// TIA Portal project "pick and place 3 things" (V16)
// Vorlageprojekt für das Buch mit Zielsystem S7-1200

(* hardware
DEVICE "S7-1200-Station_1"  S7-1200 Station
   slot 0: "Baugruppenträger_0"  Rack  V1.0
   slot 1: "PLC_1"  CPU 1211C DC/DC/DC  6ES7 211-1AE40-0XB0  V4.1
*)

// ===== PLC "PLC_1"  CPU 1211C DC/DC/DC =====

VAR_GLOBAL   // PLC tag table "Standard-Variablentabelle"
   "start" AT %I0.0 : Bool;
   "conv" AT %Q0.0 : Bool;
   "emitter" AT %Q0.1 : Bool;
   "z down" AT %Q0.2 : Bool;
   "grab" AT %Q0.3 : Bool;
   "z sensor" AT %I0.1 : Bool;
   "diffuse sens" AT %I0.2 : Bool;
   "diffuse sens memory" AT %M0.0 : Bool;
   "box detecd" AT %I0.3 : Bool;
   "box detecd memory" AT %M0.1 : Bool;
   "grab memory" AT %M0.2 : Bool;
   "z sens memory" AT %M0.3 : Bool;
   "x move" AT %Q0.4 : Bool;
   "x sensor" AT %I0.4 : Bool;
   "x sens memory\" AT %M0.4 : Bool;
   "Tag_1" AT %M0.5 : Bool;
   "Tag_2" AT %M0.7 : Bool;
   "set for timer1" AT %M1.0 : Bool;
   "Tag_4" AT %M1.1 : Bool;
   "Tag_5" AT %M1.2 : Bool;
   "set for timer 2" AT %M1.3 : Bool;
   "conv2" AT %Q0.5 : Bool;
   "diffues2" AT %I0.5 : Bool;
   "Tag_7" AT %M0.6 : Bool;
   "emitter2" AT %Q0.6 : Bool;
   "counter" AT %M1.4 : Bool;
   "Tag_9" AT %M1.5 : Bool;
   "Tag_10" AT %M1.6 : Bool;
   "Tag_8" AT %M2.0 : Bool;
   "sr for counter" AT %M2.1 : Bool;
   "reset for counter sr" AT %M2.2 : Bool;
   "stop" AT %I0.6 : Bool;
   "Tag_13" AT %M2.5 : Bool;
   "Tag_14" AT %M3.1 : Bool;
END_VAR

// folder: System blocks/Program resources

DATA_BLOCK "IEC_Timer_0_DB"   // DB1
{ S7_Optimized_Access := 'TRUE' }
AUTHOR : Simatic
FAMILY : IEC
NAME : IEC_TMR
VERSION : 1.0
// stored: InstanceOfName IEC_TIMER
"IEC_TIMER"
BEGIN
END_DATA_BLOCK

DATA_BLOCK "IEC_Timer_0_DB_1"   // DB2
{ S7_Optimized_Access := 'TRUE' }
AUTHOR : Simatic
FAMILY : IEC
NAME : IEC_TMR
VERSION : 1.0
// stored: InstanceOfName IEC_TIMER
"IEC_TIMER"
BEGIN
END_DATA_BLOCK

DATA_BLOCK "IEC_Counter_0_DB"   // DB3
{ S7_Optimized_Access := 'TRUE' }
AUTHOR : Simatic
FAMILY : IEC
NAME : CNTR
VERSION : 1.0
// stored: InstanceOfName IEC_COUNTER
"IEC_COUNTER"
BEGIN
END_DATA_BLOCK

// folder: (top level)

FUNCTION "Block_1" : Void   // FC1, LAD
{ S7_Optimized_Access := 'TRUE' }
VERSION : 0.1
   VAR_TEMP   // added for the SCL form of the ladder/FBD networks
      _w1 : Bool;
   END_VAR
BEGIN

REGION Network 1
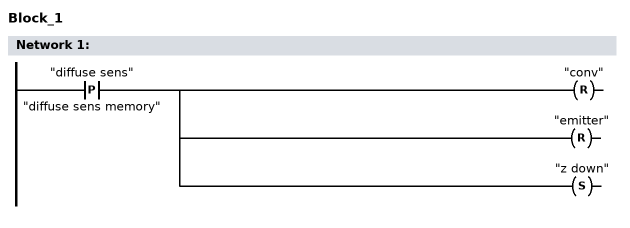
   RUNG wire#powerrail
      P_Contact(operand := "diffuse sens", bit := "diffuse sens memory")
      wire#w1
      R_Coil( "conv" )
   END_RUNG
   RUNG wire#w1
      R_Coil( "emitter" )
   END_RUNG
   RUNG wire#w1
      S_Coil( "z down" )
   END_RUNG
   // the same network as SCL:
   #_w1 := "diffuse sens" AND NOT "diffuse sens memory";   // rising edge of "diffuse sens"
   "diffuse sens memory" := "diffuse sens";
   IF #_w1 THEN
       "conv" := FALSE;
       "emitter" := FALSE;
       "z down" := TRUE;
   END_IF;
END_REGION
END_FUNCTION

FUNCTION "Block_2" : Void   // FC2, LAD
{ S7_Optimized_Access := 'TRUE' }
VERSION : 0.1
   VAR_TEMP   // added for the SCL form of the ladder/FBD networks
      _w1 : Bool;
      _w2 : Bool;
   END_VAR
BEGIN

REGION Network 1
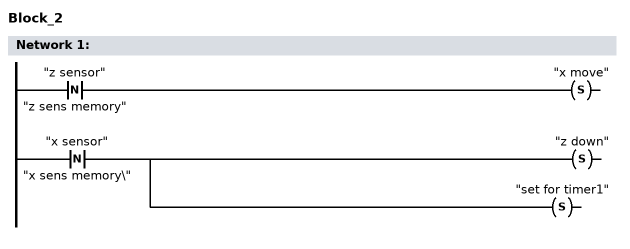
   RUNG wire#powerrail
      N_Contact(operand := "z sensor", bit := "z sens memory")
      S_Coil( "x move" )
   END_RUNG
   RUNG wire#powerrail
      N_Contact(operand := "x sensor", bit := "x sens memory\")
      wire#w1
      S_Coil( "z down" )
   END_RUNG
   RUNG wire#w1
      S_Coil( "set for timer1" )
   END_RUNG
   // the same network as SCL:
   #_w1 := NOT "z sensor" AND "z sens memory";   // falling edge of "z sensor"
   "z sens memory" := "z sensor";
   IF #_w1 THEN "x move" := TRUE; END_IF;
   #_w2 := NOT "x sensor" AND "x sens memory\";   // falling edge of "x sensor"
   "x sens memory\" := "x sensor";
   IF #_w2 THEN
       "z down" := TRUE;
       "set for timer1" := TRUE;
   END_IF;
END_REGION
END_FUNCTION

FUNCTION "MHJ-PLC-Lab-Function-S71200" : Void   // FC9000, SCL
{ S7_Optimized_Access := 'TRUE' }
VERSION : 0.1
   VAR_TEMP
      rdTimeReturn : Int;
      outputTime : DTL;
      SyncVal : Byte;
      forVal : Int;
      forVal_2 : Int;
      Value : Byte;
   END_VAR
   VAR CONSTANT
      CompVal : Byte := 16#34;
      Value_01 : Byte := 16#11;
      Value_01_DW : DWord := 16#A165_D992;
      Value_02_DW : DWord := 16#58BE_4401;
   END_VAR
BEGIN

   #Value:=PEEK(area := 16#82,
        dbNumber := 0,
        byteOffset := 511);
   #Value := #Value + 1;

   POKE(area := 16#82,
        dbNumber := 0,
        byteOffset := 511,
        value := #Value);

   POKE(area:=16#81,
        dbNumber:=0,
        byteOffset:=1016,
        value:=#Value_01_DW);
   POKE(area := 16#81,
        dbNumber := 0,
        byteOffset := 1020,
        value := #Value_02_DW);

   POKE(area := 16#81,
        dbNumber := 0,
        byteOffset := 511,
        value := B#16#00);

   FOR #forVal := 0 TO 120 DO
       FOR #forVal_2:=0 TO 10 DO
           #rdTimeReturn:=RD_SYS_T(#outputTime);
           #rdTimeReturn := WR_SYS_T(#outputTime);
           #rdTimeReturn := RD_SYS_T(#outputTime);
           #rdTimeReturn := WR_SYS_T(#outputTime);
       END_FOR;
       #SyncVal:= PEEK(area := 16#81,
                      dbNumber := 0,
                      byteOffset := 511);
       IF #SyncVal = #CompVal THEN
          GOTO M_1;
       END_IF;
   END_FOR;
   RETURN;

   M_1:
   POKE(area := 16#81,
        dbNumber := 0,
        byteOffset := 511,
        value := B#16#0);
END_FUNCTION

ORGANIZATION_BLOCK "Main"   // OB1, LAD, ProgramCycle
TITLE = "Main Program Sweep (Cycle)"
{ S7_Optimized_Access := 'TRUE' }
VERSION : 0.1
   VAR_INPUT
      Initial_Call : Bool;   // Initial call of this OB
      Remanence : Bool;   // =True, if remanent data are available
   END_VAR
   VAR_TEMP   // added for the SCL form of the ladder/FBD networks
      _w1 : Bool;
      _w2 : Bool;
   END_VAR
BEGIN

REGION Network 1
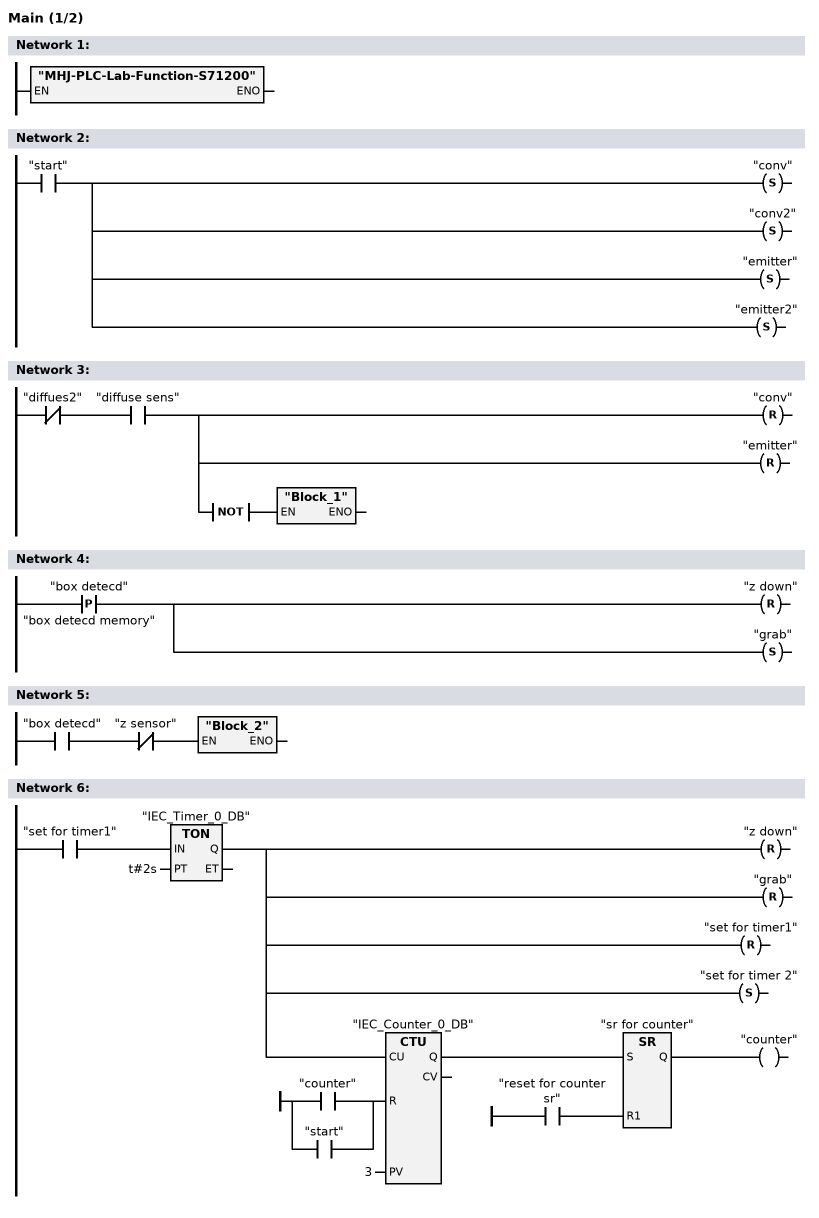
   RUNG wire#powerrail
      "MHJ-PLC-Lab-Function-S71200"()
   END_RUNG
   // the same network as SCL:
   "MHJ-PLC-Lab-Function-S71200"();
END_REGION

REGION Network 2
   RUNG wire#powerrail
      Contact( "start" )
      wire#w1
      S_Coil( "conv" )
   END_RUNG
   RUNG wire#w1
      S_Coil( "conv2" )
   END_RUNG
   RUNG wire#w1
      S_Coil( "emitter" )
   END_RUNG
   RUNG wire#w1
      S_Coil( "emitter2" )
   END_RUNG
   // the same network as SCL:
   IF "start" THEN
       "conv" := TRUE;
       "conv2" := TRUE;
       "emitter" := TRUE;
       "emitter2" := TRUE;
   END_IF;
END_REGION

REGION Network 3
   RUNG wire#powerrail
      I_Contact( "diffues2" )
      Contact( "diffuse sens" )
      wire#w1
      R_Coil( "conv" )
   END_RUNG
   RUNG wire#w1
      R_Coil( "emitter" )
   END_RUNG
   RUNG wire#w1
      Not()
      "Block_1"()
   END_RUNG
   // the same network as SCL:
   #_w1 := NOT "diffues2" AND "diffuse sens";
   IF #_w1 THEN
       "conv" := FALSE;
       "emitter" := FALSE;
   END_IF;
   IF NOT #_w1 THEN "Block_1"(); END_IF;
END_REGION

REGION Network 4
   RUNG wire#powerrail
      P_Contact(operand := "box detecd", bit := "box detecd memory")
      wire#w1
      R_Coil( "z down" )
   END_RUNG
   RUNG wire#w1
      S_Coil( "grab" )
   END_RUNG
   // the same network as SCL:
   #_w1 := "box detecd" AND NOT "box detecd memory";   // rising edge of "box detecd"
   "box detecd memory" := "box detecd";
   IF #_w1 THEN
       "z down" := FALSE;
       "grab" := TRUE;
   END_IF;
END_REGION

REGION Network 5
   RUNG wire#powerrail
      Contact( "box detecd" )
      I_Contact( "z sensor" )
      "Block_2"()
   END_RUNG
   // the same network as SCL:
   IF "box detecd" AND NOT "z sensor" THEN "Block_2"(); END_IF;
END_REGION

REGION Network 6
   "IEC_Timer_0_DB".TON(IN := "set for timer1", PT := t#2s);
   IF "IEC_Timer_0_DB".Q THEN
       "z down" := FALSE;
       "grab" := FALSE;
       "set for timer1" := FALSE;
       "set for timer 2" := TRUE;
   END_IF;
   "IEC_Counter_0_DB".CTU(CU := "IEC_Timer_0_DB".Q, R := "counter" OR "start", PV := 3);
   IF "IEC_Counter_0_DB".Q THEN
       "sr for counter" := TRUE;   // SR flip-flop
   END_IF;
   IF "reset for counter sr" THEN "sr for counter" := FALSE; END_IF;
   "counter" := "sr for counter";
END_REGION

REGION Network 7
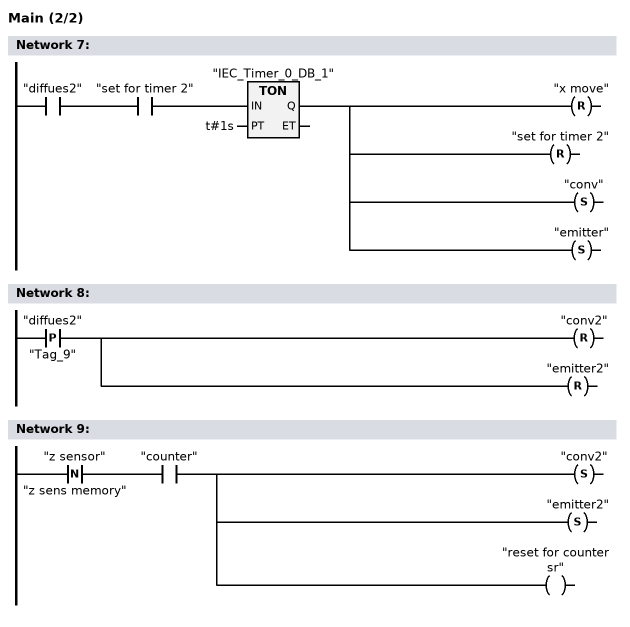
   "IEC_Timer_0_DB_1".TON(IN := "diffues2" AND "set for timer 2", PT := t#1s);
   IF "IEC_Timer_0_DB_1".Q THEN
       "x move" := FALSE;
       "set for timer 2" := FALSE;
       "conv" := TRUE;
       "emitter" := TRUE;
   END_IF;
END_REGION

REGION Network 8
   RUNG wire#powerrail
      P_Contact(operand := "diffues2", bit := "Tag_9")
      wire#w1
      R_Coil( "conv2" )
   END_RUNG
   RUNG wire#w1
      R_Coil( "emitter2" )
   END_RUNG
   // the same network as SCL:
   #_w1 := "diffues2" AND NOT "Tag_9";   // rising edge of "diffues2"
   "Tag_9" := "diffues2";
   IF #_w1 THEN
       "conv2" := FALSE;
       "emitter2" := FALSE;
   END_IF;
END_REGION

REGION Network 9
   RUNG wire#powerrail
      N_Contact(operand := "z sensor", bit := "z sens memory")
      Contact( "counter" )
      wire#w1
      S_Coil( "conv2" )
   END_RUNG
   RUNG wire#w1
      S_Coil( "emitter2" )
   END_RUNG
   RUNG wire#w1
      Coil( "reset for counter sr" )
   END_RUNG
   // the same network as SCL:
   #_w1 := NOT "z sensor" AND "z sens memory";   // falling edge of "z sensor"
   "z sens memory" := "z sensor";
   #_w2 := #_w1 AND "counter";
   IF #_w2 THEN
       "conv2" := TRUE;
       "emitter2" := TRUE;
   END_IF;
   "reset for counter sr" := #_w2;
END_REGION
END_ORGANIZATION_BLOCK